(* PLC project x *)

FUNCTION_BLOCK LD_MISC
  VAR_INPUT
    xA : BOOL;
  END_VAR
  VAR  (* added by the conversion: wires and edge detectors of the diagram *)
    R_TRIG1 : R_TRIG;
    R_TRIG2 : R_TRIG;
    R_TRIG3 : R_TRIG;
    _ADD15_ENO : BOOL;
    _ADD15_OUT : ANY;
  END_VAR

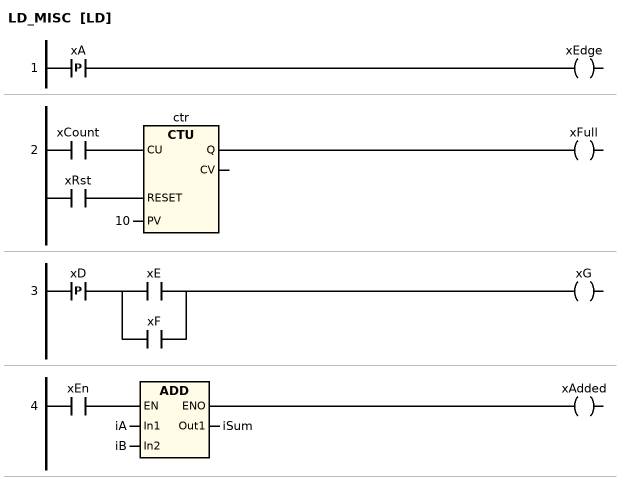
(* LD diagram, written out as Structured Text *)
R_TRIG1(CLK := NOT xA);
xEdge := R_TRIG1.Q;
R_TRIG2(CLK := xCount);
ctr(CU := R_TRIG2.Q, RESET := xRst, PV := 10);
xFull := ctr.Q;
R_TRIG3(CLK := xD);
xG := R_TRIG3.Q AND (xE OR xF);
_ADD15_OUT := ADD(EN := xEn, IN1 := iA, IN2 := iB, ENO => _ADD15_ENO);
xAdded := _ADD15_ENO;
IF _ADD15_ENO THEN iSum := _ADD15_OUT; END_IF;
END_FUNCTION_BLOCK
